// TIA Portal V19 export
TYPE "LUC_typeButtons"
TITLE = LUC_typeButtons
// Properties of  HMI buttons configured from the PLC
// stored: Access Published
   STRUCT
      visibility { ExternalWritable := 'False'} : Word;   // Sets the visibility property in the buttons of the HMI
      operatorControlAllowed { ExternalWritable := 'False'} : Word;   // Sets the operator control allowed property in the buttons of the HMI
      active { ExternalWritable := 'False'} : Word;   // Sets the alternative border color property in the buttons of the HMI
   END_STRUCT;
END_TYPE
